FUNCTION_BLOCK FB_TrafficLight
VAR
    state : INT;  // 0=Red, 1=RedAmber, 2=Green, 3=Amber
END_VAR

METHOD Step : INT
CASE state OF
    0:
        state := 1;
    1:
        state := 2;
    2:
        state := 0;
    3:
        state := 0;
END_CASE;
Step := state;
END_METHOD

END_FUNCTION_BLOCK

(* stored: Version 1.1.0.1
   POU FB_TrafficLight: Id {bbc8da29-dd17-49fe-bb76-9cd6f8ed87f1}, SpecialFunc None
   Method Step: Id {97346fe1-2487-4375-a092-e1400fbe85ab} *)
